RESOURCE_TYPE top
  (* Standard: 61499-2 *)
  (* Version 0.1, 2017-00-25, hpea485, UOA *)
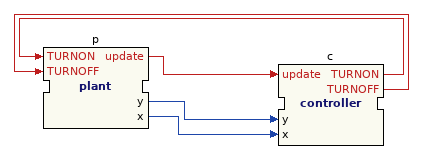
  FBS
    p : plant;
    c : controller;
  END_FBS
  EVENT_CONNECTIONS
    p.update TO c.update;
    c.TURNON TO p.TURNON;
    c.TURNOFF TO p.TURNOFF;
  END_CONNECTIONS
  DATA_CONNECTIONS
    p.y TO c.y;
    p.x TO c.x;
  END_CONNECTIONS
END_RESOURCE_TYPE
